// Mitsubishi GX Works2 project: yudomotmutistep   PLC: Q03UDV

PROGRAM MAIN
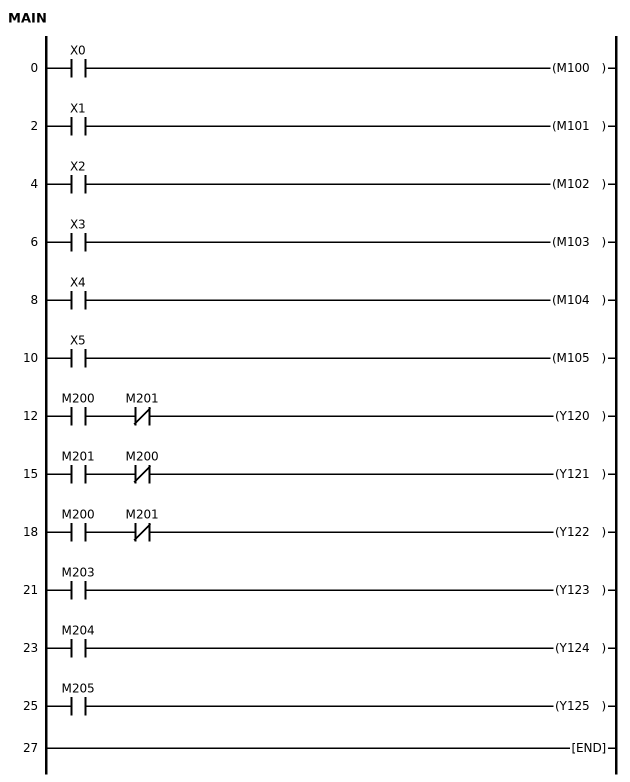
0     LD      X0
      OUT     M100
2     LD      X1
      OUT     M101
4     LD      X2
      OUT     M102
6     LD      X3
      OUT     M103
8     LD      X4
      OUT     M104
10    LD      X5
      OUT     M105
12    LD      M200
      ANI     M201
      OUT     Y120
15    LD      M201
      ANI     M200
      OUT     Y121
18    LD      M200
      ANI     M201
      OUT     Y122
21    LD      M203
      OUT     Y123
23    LD      M204
      OUT     Y124
25    LD      M205
      OUT     Y125
27    END
END_PROGRAM
